// TIA Portal project "运动控制项目" (V20)

(* hardware
DEVICE "S7-1200 station_1"  S7-1200 Station
   slot 0: "Rack_0"  S7-1200 Rack  Rack  V1.0
   slot 1: "PLC_1"  CPU 1215C DC/DC/DC  6ES7 215-1AG40-0XB0  V4.6
   slot 3: "CB 1241 (RS485)"  CB 1241 (RS485)  6ES7 241-1CH30-1XB0  V1.0
*)

// ===== PLC "PLC_1"  CPU 1215C DC/DC/DC =====

VAR_GLOBAL   // PLC tag table "默认变量表"
   "System_Byte" AT %MB1 : Byte;
   "FirstScan" AT %M1.0 : Bool;
   "DiagStatusUpdate" AT %M1.1 : Bool;
   "AlwaysTRUE" AT %M1.2 : Bool;
   "AlwaysFALSE" AT %M1.3 : Bool;
   "Clock_Byte" AT %MB0 : Byte;
   "Clock_10Hz" AT %M0.0 : Bool;
   "Clock_5Hz" AT %M0.1 : Bool;
   "Clock_2.5Hz" AT %M0.2 : Bool;
   "Clock_2Hz" AT %M0.3 : Bool;
   "Clock_1.25Hz" AT %M0.4 : Bool;
   "Clock_1Hz" AT %M0.5 : Bool;
   "Clock_0.625Hz" AT %M0.6 : Bool;
   "Clock_0.5Hz" AT %M0.7 : Bool;
   "Tag_1" AT %Q0.6 : Bool;
   "Tag_2" AT %I0.3 : Bool;
   "Tag_3" AT %I0.4 : Bool;
   "Tag_4" AT %I0.5 : Bool;
   "Tag_5" AT %I0.6 : Bool;
   "Tag_6" AT %I0.7 : Bool;
   "Tag_7" AT %M2.4 : Bool;
   "Tag_8" AT %M2.5 : Bool;
END_VAR

VAR_GLOBAL   // PLC tag table "input"
   "limit_left" AT %I0.0 : Bool;
   "stop" AT %I0.1 : Bool;
   "limit_right" AT %I0.2 : Bool;
   "Tag_9" AT %I0.3 : Bool;
END_VAR

VAR_GLOBAL   // PLC tag table "output"
   "puls_plus" AT %Q0.0 : Bool;
   "red_w" AT %Q0.1 : Bool;
   "dir_plus" AT %Q0.2 : Bool;
   "green_s" AT %Q0.3 : Bool;
   "red_s" AT %Q0.4 : Bool;
   "yellow_s" AT %Q0.5 : Bool;
END_VAR

VAR_GLOBAL   // PLC tag table "intermedia"
   "cnt" AT %MB5 : Byte;
   "p1" AT %M2.0 : Bool;
   "p2" AT %M2.1 : Bool;
   "activate_x" AT %M2.2 : Bool;
   "ready_x" AT %M2.3 : Bool;
END_VAR

DATA_BLOCK "丝杠运动控制测试数据块_1"   // DB4
{ S7_Optimized_Access := 'TRUE' }
VERSION : 0.1
// stored: InstanceOfName 丝杠运动控制测试
"丝杠运动控制测试"
BEGIN
END_DATA_BLOCK

DATA_BLOCK "喷泉fc"   // DB5
{ S7_Optimized_Access := 'TRUE' }
VERSION : 0.1
BEGIN
END_DATA_BLOCK

// folder: 作业

DATA_BLOCK "交通红绿灯_流程SCL_DB"   // DB2
{ S7_Optimized_Access := 'TRUE' }
VERSION : 0.1
// stored: InstanceOfName 交通红绿灯_流程SCL
"交通红绿灯_流程SCL"
BEGIN
END_DATA_BLOCK

DATA_BLOCK "交通红绿灯_比较SCL_DB"   // DB3
{ S7_Optimized_Access := 'TRUE' }
VERSION : 0.1
// stored: InstanceOfName 交通红绿灯_比较SCL
"交通红绿灯_比较SCL"
BEGIN
END_DATA_BLOCK

// folder: (top level)

DATA_BLOCK "桌面丝杠"   // DB1, Motion_DB
{ S7_Optimized_Access := 'TRUE' }
AUTHOR : SIMATIC
FAMILY : BasicMC
NAME : TO_PosAx
VERSION : 8.0
// stored: InstanceOfName TO_PositioningAxis
"TO_PositioningAxis"
BEGIN
   // Axis.EnableOutput_AddressCU = %M2.2
   // Axis.PassiveHomingReferencePointSwitch_AddressCU = %I0.1
   // Axis.HomingReferencePointSwitch_AddressCU = %I0.1
   // Axis.PositionLimitsMin_AddressCU = %I0.0
   // Axis.PositionLimitsMax_AddressCU = %I0.2
   // Axis.OnlinePtoModeCU = 16#0000_0002
   // Axis.DirectionOutputEnabledCU = TRUE
   // Axis.SelectedChannel2EnumCU = %Q0.2
   // Axis.SelectedChannel1EnumCU = %Q0.0
   // Pulse.MinDeltaDeltaFrequencyCU = 0.004
   // Pulse.MaxDeltaDeltaFrequencyCU = 1.0E+10
   // Pulse.MinDeltaFrequencyCU = 0.005
   // Pulse.MaxDeltaFrequencyCU = 9.5E+9
   // Pulse.MinFrequencyCU = 1.0
   // Pulse.MaxFrequencyCU = 100000.0
   // Pulse.OutputSourceCU = 16#0000_0000
   // Axis.SelectPTO = 0
END_DATA_BLOCK

FUNCTION_BLOCK "丝杠运动控制测试"   // FB1, LAD
{ S7_Optimized_Access := 'TRUE' }
VERSION : 0.1
   VAR
      if_done : Bool;
      if_error : Bool;
      if_busy : Bool;
      error_id : Word;
      error_info : Word;
      ativate_x : Bool;
      ready_x : Bool;
      run_axis_x : Bool;
      position_x : DInt;
      MC_Power_Instance : MC_Power;
      MC_Home_Instance : MC_Home;
      MC_Power_Instance_1 : MC_Power;
      MC_ReadParam_Instance : MC_ReadParam;
      MC_WriteParam_Instance : MC_WriteParam;
      MC_MoveAbsolute_Instance : MC_MoveAbsolute;
      MC_MoveJog_Instance : MC_MoveJog;
      MC_Reset_Instance : MC_Reset;
   END_VAR
BEGIN

REGION Network 1
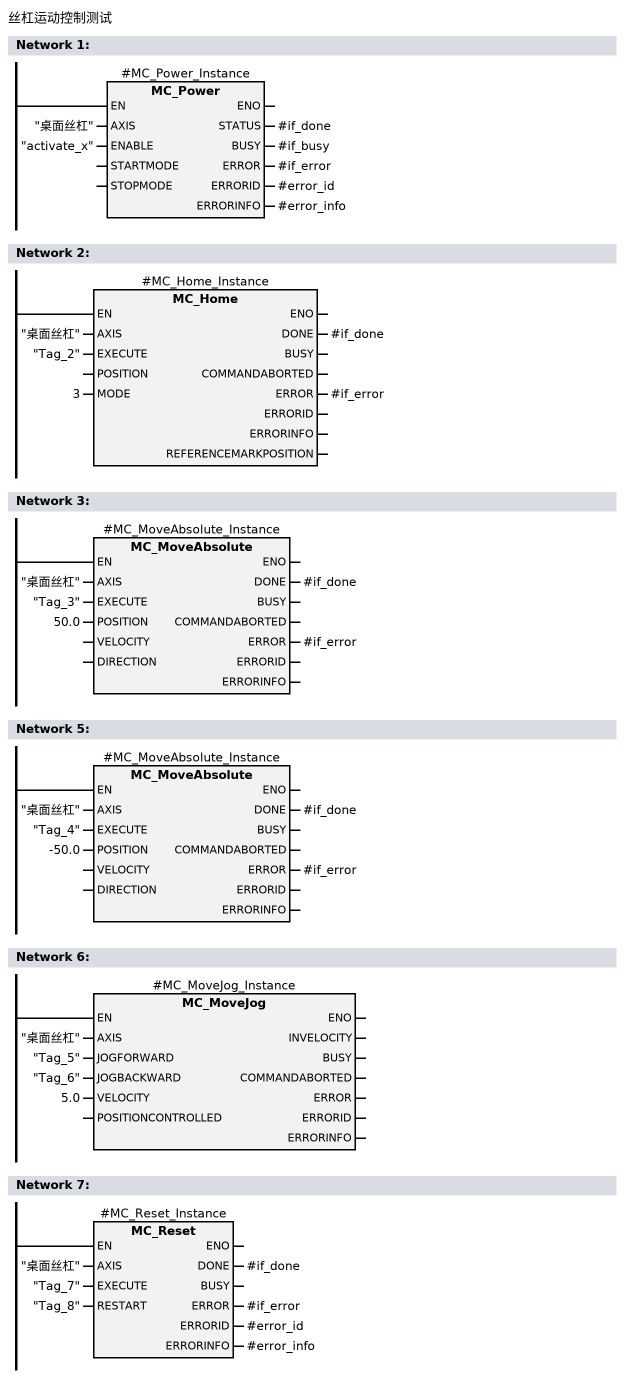
   #MC_Power_Instance(Axis := "桌面丝杠",   // MC_Power
                      Enable := "activate_x",
                      Status => #if_done,
                      Busy => #if_busy,
                      Error => #if_error,
                      ErrorID => #error_id,
                      ErrorInfo => #error_info);
END_REGION

REGION Network 2
   #MC_Home_Instance(Axis := "桌面丝杠", Execute := "Tag_2", Mode := 3, Done => #if_done, Error => #if_error);   // MC_Home
END_REGION

REGION Network 3
   #MC_MoveAbsolute_Instance(Axis := "桌面丝杠",   // MC_MoveAbsolute
                           Execute := "Tag_3",
                           Position := 50.0,
                           Done => #if_done,
                           Error => #if_error);
END_REGION

REGION Network 5
   #MC_MoveAbsolute_Instance(Axis := "桌面丝杠",   // MC_MoveAbsolute
                           Execute := "Tag_4",
                           Position := -50.0,
                           Done => #if_done,
                           Error => #if_error);
END_REGION

REGION Network 6
   #MC_MoveJog_Instance(Axis := "桌面丝杠", JogForward := "Tag_5", JogBackward := "Tag_6", Velocity := 5.0);   // MC_MoveJog
END_REGION

REGION Network 7
   #MC_Reset_Instance(Axis := "桌面丝杠",   // MC_Reset
                      Execute := "Tag_7",
                      Restart := "Tag_8",
                      Done => #if_done,
                      Error => #if_error,
                      ErrorID => #error_id,
                      ErrorInfo => #error_info);
END_REGION
END_FUNCTION_BLOCK

FUNCTION "喷泉项目" : Void   // FC2, LAD
{ S7_Optimized_Access := 'TRUE' }
VERSION : 0.1
BEGIN
END_FUNCTION

ORGANIZATION_BLOCK "Main"   // OB1, LAD, ProgramCycle
TITLE = "Main Program Sweep (Cycle)"
{ S7_Optimized_Access := 'TRUE' }
VERSION : 0.1
   VAR_INPUT
      Initial_Call : Bool;   // Initial call of this OB
      Remanence : Bool;   // =True, if remanent data are available
   END_VAR
BEGIN

REGION Network 1 (SCL)
   (*



   *)
END_REGION

REGION Network 2
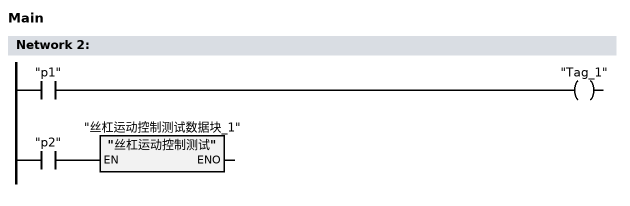
   RUNG wire#powerrail
      Contact( "p1" )
      Coil( "Tag_1" )
   END_RUNG
   RUNG wire#powerrail
      Contact( "p2" )
      "丝杠运动控制测试数据块_1"()
   END_RUNG
   // the same network as SCL:
   "Tag_1" := "p1";
   IF "p2" THEN
       "丝杠运动控制测试数据块_1"();   // "丝杠运动控制测试"
   END_IF;
END_REGION
END_ORGANIZATION_BLOCK

// folder: 作业

FUNCTION_BLOCK "交通红绿灯_流程SCL"   // FB2, LAD
{ S7_Optimized_Access := 'TRUE' }
VERSION : 0.1
   VAR
      start_pressed_trig : R_TRIG;
      stop_pressed_trig : R_TRIG;
      start_trig : R_TRIG;
      started : Bool;
      stoped : Bool;
      step_w : Byte;
      step_s : Byte;
      Timer_0 : TON_TIME;
      Timer_1 : TON_TIME;
      Timer_2 : TON_TIME;
      Timer_3 : TON_TIME;
      time_w : Time;
      time_s : Time;
   END_VAR
BEGIN

REGION Network 2 (SCL)
   IF "FirstScan" THEN
       #started := #stoped := 0;
       #step_w := #step_s := 0;
   END_IF;

   //initiate
   #start_pressed_trig(CLK := "limit_left");
   #stop_pressed_trig(CLK := "stop");
   #start_trig(CLK := #started);

   #Timer_0(IN := #started, PT := #time_w);
   #Timer_1(IN := #started, PT := #time_s);
   #Timer_2(IN := "AlwaysTRUE", PT := t#500ms);
   #Timer_3(IN := #Timer_2.Q,PT := t#500ms);
   IF #Timer_3.Q THEN
       RESET_TIMER(#Timer_2);
   END_IF;

   IF #start_pressed_trig.Q THEN
       #started := 1;
       #stoped := 0;
   END_IF;

   IF #start_trig.Q THEN
       #stoped := 0;
       #step_s := #step_w := 0;
       "green_s" := "puls_plus" := "dir_plus" := "yellow_s" := "red_w" := "red_s" := 0;
       #time_w := t#5s;
       #time_s := t#10s;
       RESET_TIMER(#Timer_0);
       RESET_TIMER(#Timer_1);
   END_IF;

   IF #stop_pressed_trig.Q THEN
       #stoped := 1;
   END_IF;

   IF #started THEN
       //东西向
       IF #step_w = 0 THEN
           "puls_plus" := 1;
           IF #Timer_0.Q THEN
               "puls_plus" := 0;
               RESET_TIMER(#Timer_0);
               #time_w := T#3s;
               #step_w += 1;
           END_IF;
       END_IF;

       IF #step_w = 1 THEN
           "puls_plus" := #Timer_2.Q;
           IF #Timer_0.Q THEN
               "puls_plus" := 0;
               RESET_TIMER(#Timer_0);
               #time_w := T#2s;
               #step_w += 1;
           END_IF;
       END_IF;

       IF #step_w = 2 THEN
           "dir_plus" := 1;
           IF #Timer_0.Q THEN
               "dir_plus" := 0;
               RESET_TIMER(#Timer_0);
               #time_w := T#10s;
               #step_w += 1;
           END_IF;
       END_IF;

       IF #step_w = 3 THEN
           "red_w":= 1;
           IF #Timer_0.Q THEN
               "red_w" := 0;
               RESET_TIMER(#Timer_0);
               #time_w := T#5s;
               #step_w := 0;
           END_IF;
       END_IF;

       //南北向
       IF #step_s = 0 THEN
           "red_s" := 1;
           IF #Timer_1.Q THEN
               "red_s" := 0;
               RESET_TIMER(#Timer_1);
               #time_s := T#5s;
               #step_s += 1;
           END_IF;
       END_IF;

       IF #step_s = 1 THEN
           "green_s" := 1;
           IF #Timer_1.Q THEN
               "green_s" := 0;
               RESET_TIMER(#Timer_1);
               #time_s := T#3s;
               #step_s += 1;
           END_IF;
       END_IF;

       IF #step_s = 2 THEN
          "green_s" := #Timer_2.Q;
          IF #Timer_1.Q THEN
              "green_s" := 0;
               RESET_TIMER(#Timer_1);
               #time_s := T#2s;
               #step_s += 1;
           END_IF;
       END_IF;

       IF #step_s = 3 THEN
           "yellow_s" := 1;
           IF #Timer_1.Q THEN
               "yellow_s" := 0;
               RESET_TIMER(#Timer_1);
               #time_s := T#10s;
               #step_s := 0;
               #step_w := 0;
               "red_w" := 0;
               RESET_TIMER(#Timer_0);
               #time_w := T#5s;
               #step_w := 0;

               IF #stoped THEN
                   #started := 0;
                   #stoped := 0;
               END_IF;
           END_IF;
       END_IF;
   END_IF;

   IF NOT #stoped AND NOT #started THEN
       "yellow_s" := #Timer_2.Q;
       "dir_plus" := #Timer_2.Q;
   END_IF;
END_REGION
END_FUNCTION_BLOCK

FUNCTION_BLOCK "交通红绿灯_比较SCL"   // FB3, LAD
{ S7_Optimized_Access := 'TRUE' }
VERSION : 0.1
   VAR
      start_pressed_trig : R_TRIG;
      stop_pressed_trig : R_TRIG;
      start_trig : R_TRIG;
      started : Bool;
      stoped : Bool;
      step_w : Byte;
      step_s : Byte;
      Timer_0 : TON_TIME;
      Timer_1 : TON_TIME;
      Timer_2 : TON_TIME;
      Timer_3 : TON_TIME;
      time_w : Time;
      time_s : Time;
      button : Array[0..10] of Bool;
      b1 : Bool;
      b2 : Bool;
      b4 : Bool;
      b3 : Bool;
      b5 : Bool;
   END_VAR
BEGIN

REGION Network 2 (SCL)
   IF "FirstScan" THEN
       #started := #stoped := 0;
       #step_w := #step_s := 0;
   END_IF;

   //initiate
   #start_pressed_trig(CLK := "limit_left");
   #stop_pressed_trig(CLK := "stop");
   #start_trig(CLK := #started);

   #Timer_0(IN := #started, PT := t#20S);
   #Timer_2(IN := "AlwaysTRUE", PT := t#500ms);
   #Timer_3(IN := #Timer_2.Q,PT := t#500ms);
   IF #Timer_3.Q THEN
       RESET_TIMER(#Timer_2);
   END_IF;

   IF #start_pressed_trig.Q THEN
       #started := 1;
       #stoped := 0;
   END_IF;

   IF #start_trig.Q THEN
       #stoped := 0;
       RESET_TIMER(#Timer_0);
       RESET_TIMER(#Timer_2);
   END_IF;

   IF #stop_pressed_trig.Q THEN
       #stoped := 1;
   END_IF;

   IF #started THEN
       //东西向
       "puls_plus" := #Timer_0.ET > t#0s AND #Timer_0.ET <= t#5s OR (#Timer_0.ET > t#5s AND #Timer_0.ET <= t#8s AND #Timer_2.Q);
       "dir_plus" := #Timer_0.ET > t#8s AND #Timer_0.ET <= t#10s;
       "red_w" := #Timer_0.ET > t#10s AND #Timer_0.ET <= t#20s;

       //南北向
       "red_s" := #Timer_0.ET > t#0s AND #Timer_0.ET <= t#10s;
       "green_s" := #Timer_0.ET > t#10s AND #Timer_0.ET <= t#13s OR (#Timer_0.ET > t#13s AND #Timer_0.ET <= t#15s AND #Timer_2.Q);
       "yellow_s" := #Timer_0.ET > t#15s AND #Timer_0.ET < t#20s;

       IF #Timer_0.ET >= t#20S THEN
           RESET_TIMER(#Timer_0);
           RESET_TIMER(#Timer_1);

           #started := NOT #stoped;
           #stoped := 0;
       END_IF;
   END_IF;

   IF NOT #stoped AND NOT #started THEN
       "green_s" := "puls_plus" := "red_s" := "red_w" := 0;
       "yellow_s" := #Timer_2.Q;
       "dir_plus" := #Timer_2.Q;
   END_IF;
END_REGION
END_FUNCTION_BLOCK

FUNCTION "红绿灯_FC" : Void   // FC1, LAD
{ S7_Optimized_Access := 'TRUE' }
VERSION : 0.1
   VAR_TEMP   // added for the SCL form of the ladder/FBD networks
      _w1 : Bool;
      _w2 : Bool;
      _w3 : Bool;
   END_VAR
BEGIN

REGION Network 1
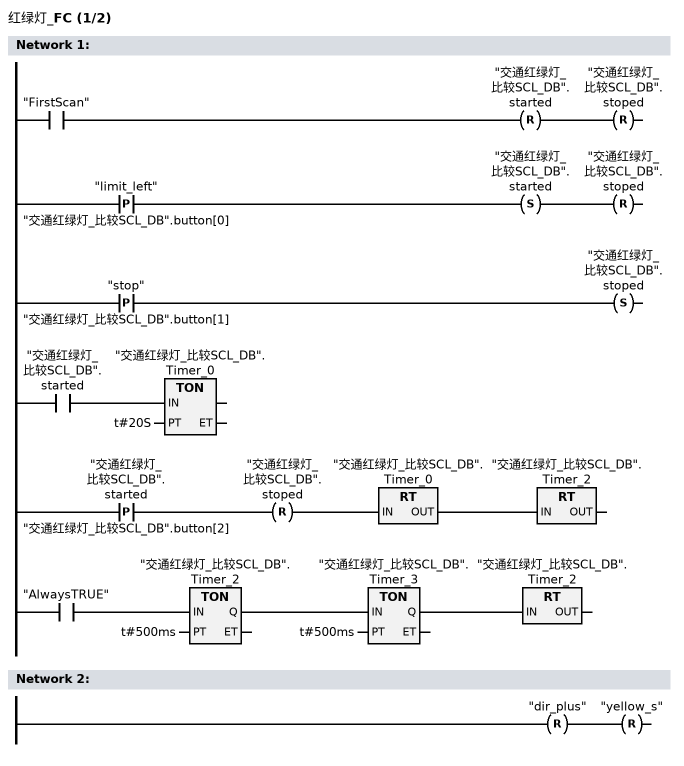
   IF "FirstScan" THEN
       "交通红绿灯_比较SCL_DB".started := FALSE;
       "交通红绿灯_比较SCL_DB".stoped := FALSE;
   END_IF;
   #_w1 := "limit_left" AND NOT "交通红绿灯_比较SCL_DB".button[0];   // rising edge of "limit_left"
   "交通红绿灯_比较SCL_DB".button[0] := "limit_left";
   IF #_w1 THEN
       "交通红绿灯_比较SCL_DB".started := TRUE;
       "交通红绿灯_比较SCL_DB".stoped := FALSE;
   END_IF;
   #_w2 := "stop" AND NOT "交通红绿灯_比较SCL_DB".button[1];   // rising edge of "stop"
   "交通红绿灯_比较SCL_DB".button[1] := "stop";
   IF #_w2 THEN "交通红绿灯_比较SCL_DB".stoped := TRUE; END_IF;
   "交通红绿灯_比较SCL_DB".Timer_0.TON(IN := "交通红绿灯_比较SCL_DB".started, PT := t#20S);
   #_w3 := "交通红绿灯_比较SCL_DB".started AND NOT "交通红绿灯_比较SCL_DB".button[2];   // rising edge of "交通红绿灯_比较SCL_DB".started
   "交通红绿灯_比较SCL_DB".button[2] := "交通红绿灯_比较SCL_DB".started;
   IF #_w3 THEN
       "交通红绿灯_比较SCL_DB".stoped := FALSE;
       RESET_TIMER("交通红绿灯_比较SCL_DB".Timer_0);
       RESET_TIMER("交通红绿灯_比较SCL_DB".Timer_2);
   END_IF;
   "交通红绿灯_比较SCL_DB".Timer_2.TON(IN := "AlwaysTRUE", PT := t#500ms);
   "交通红绿灯_比较SCL_DB".Timer_3.TON(IN := "交通红绿灯_比较SCL_DB".Timer_2.Q, PT := t#500ms);
   IF "交通红绿灯_比较SCL_DB".Timer_3.Q THEN RESET_TIMER("交通红绿灯_比较SCL_DB".Timer_2); END_IF;
END_REGION

REGION Network 2
   RUNG wire#powerrail
      R_Coil( "dir_plus" )
      R_Coil( "yellow_s" )
   END_RUNG
   // the same network as SCL:
   "dir_plus" := FALSE;
   "yellow_s" := FALSE;
END_REGION

REGION Network 3
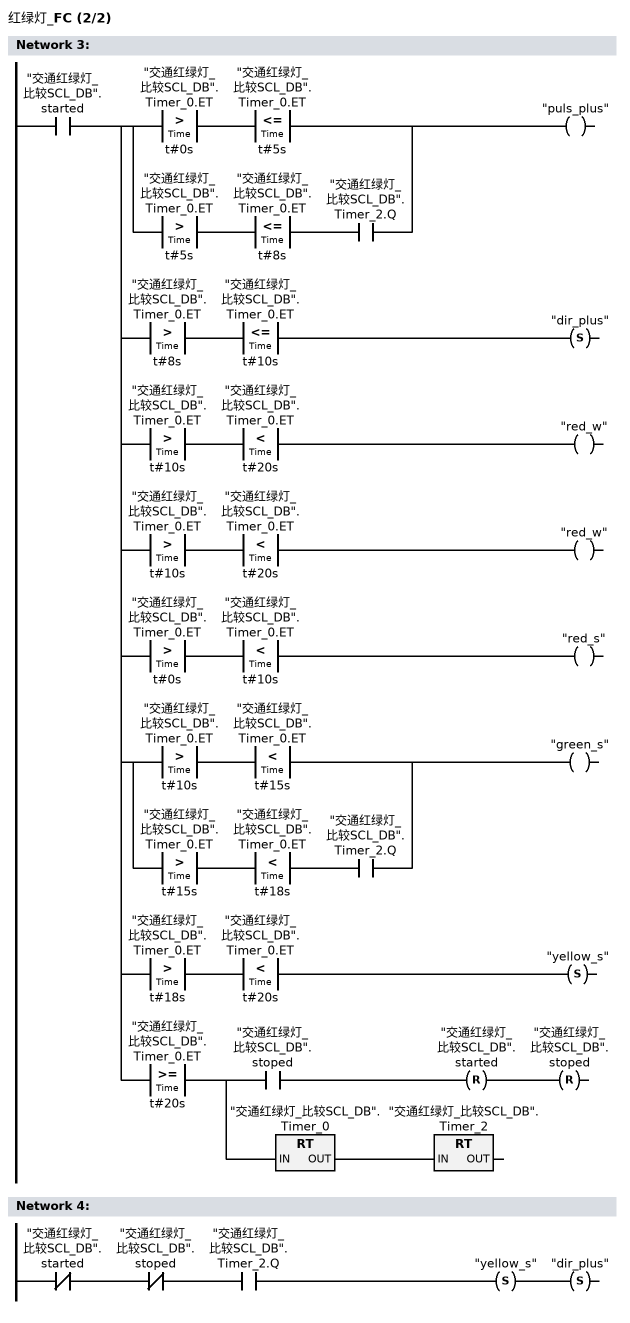
   RUNG wire#powerrail
      Contact( "交通红绿灯_比较SCL_DB".started )
      wire#w1
      { S7_Templates := "SrcType := Time" } GT_Contact(in1 := "交通红绿灯_比较SCL_DB".Timer_0.ET, in2 := t#0s)
      { S7_Templates := "SrcType := Time" } LE_Contact(in1 := "交通红绿灯_比较SCL_DB".Timer_0.ET, in2 := t#5s)
      wire#w2
      Coil( "puls_plus" )
   END_RUNG
   RUNG wire#w1
      { S7_Templates := "SrcType := Time" } GT_Contact(in1 := "交通红绿灯_比较SCL_DB".Timer_0.ET, in2 := t#5s)
      { S7_Templates := "SrcType := Time" } LE_Contact(in1 := "交通红绿灯_比较SCL_DB".Timer_0.ET, in2 := t#8s)
      Contact( "交通红绿灯_比较SCL_DB".Timer_2.Q )
   END_RUNG wire#w2
   RUNG wire#w1
      { S7_Templates := "SrcType := Time" } GT_Contact(in1 := "交通红绿灯_比较SCL_DB".Timer_0.ET, in2 := t#8s)
      { S7_Templates := "SrcType := Time" } LE_Contact(in1 := "交通红绿灯_比较SCL_DB".Timer_0.ET, in2 := t#10s)
      S_Coil( "dir_plus" )
   END_RUNG
   RUNG wire#w1
      { S7_Templates := "SrcType := Time" } GT_Contact(in1 := "交通红绿灯_比较SCL_DB".Timer_0.ET, in2 := t#10s)
      { S7_Templates := "SrcType := Time" } LT_Contact(in1 := "交通红绿灯_比较SCL_DB".Timer_0.ET, in2 := t#20s)
      Coil( "red_w" )
   END_RUNG
   RUNG wire#w1
      { S7_Templates := "SrcType := Time" } GT_Contact(in1 := "交通红绿灯_比较SCL_DB".Timer_0.ET, in2 := t#10s)
      { S7_Templates := "SrcType := Time" } LT_Contact(in1 := "交通红绿灯_比较SCL_DB".Timer_0.ET, in2 := t#20s)
      Coil( "red_w" )
   END_RUNG
   RUNG wire#w1
      { S7_Templates := "SrcType := Time" } GT_Contact(in1 := "交通红绿灯_比较SCL_DB".Timer_0.ET, in2 := t#0s)
      { S7_Templates := "SrcType := Time" } LT_Contact(in1 := "交通红绿灯_比较SCL_DB".Timer_0.ET, in2 := t#10s)
      Coil( "red_s" )
   END_RUNG
   RUNG wire#w1
      { S7_Templates := "SrcType := Time" } GT_Contact(in1 := "交通红绿灯_比较SCL_DB".Timer_0.ET, in2 := t#10s)
      { S7_Templates := "SrcType := Time" } LT_Contact(in1 := "交通红绿灯_比较SCL_DB".Timer_0.ET, in2 := t#15s)
      wire#w3
      Coil( "green_s" )
   END_RUNG
   RUNG wire#w1
      { S7_Templates := "SrcType := Time" } GT_Contact(in1 := "交通红绿灯_比较SCL_DB".Timer_0.ET, in2 := t#15s)
      { S7_Templates := "SrcType := Time" } LT_Contact(in1 := "交通红绿灯_比较SCL_DB".Timer_0.ET, in2 := t#18s)
      Contact( "交通红绿灯_比较SCL_DB".Timer_2.Q )
   END_RUNG wire#w3
   RUNG wire#w1
      { S7_Templates := "SrcType := Time" } GT_Contact(in1 := "交通红绿灯_比较SCL_DB".Timer_0.ET, in2 := t#18s)
      { S7_Templates := "SrcType := Time" } LT_Contact(in1 := "交通红绿灯_比较SCL_DB".Timer_0.ET, in2 := t#20s)
      S_Coil( "yellow_s" )
   END_RUNG
   RUNG wire#w1
      { S7_Templates := "SrcType := Time" } GE_Contact(in1 := "交通红绿灯_比较SCL_DB".Timer_0.ET, in2 := t#20s)
      wire#w4
      Contact( "交通红绿灯_比较SCL_DB".stoped )
      R_Coil( "交通红绿灯_比较SCL_DB".started )
      R_Coil( "交通红绿灯_比较SCL_DB".stoped )
   END_RUNG
   RUNG wire#w4
      RT_Coil( "交通红绿灯_比较SCL_DB".Timer_0 )
      RT_Coil( "交通红绿灯_比较SCL_DB".Timer_2 )
   END_RUNG
   // the same network as SCL:
   "puls_plus" := "交通红绿灯_比较SCL_DB".started AND ((("交通红绿灯_比较SCL_DB".Timer_0.ET > t#0s) AND ("交通红绿灯_比较SCL_DB".Timer_0.ET <= t#5s)) OR (("交通红绿灯_比较SCL_DB".Timer_0.ET > t#5s) AND ("交通红绿灯_比较SCL_DB".Timer_0.ET <= t#8s) AND "交通红绿灯_比较SCL_DB".Timer_2.Q));
   IF "交通红绿灯_比较SCL_DB".started AND ("交通红绿灯_比较SCL_DB".Timer_0.ET > t#8s) AND ("交通红绿灯_比较SCL_DB".Timer_0.ET <= t#10s) THEN
       "dir_plus" := TRUE;
   END_IF;
   "red_w" := "交通红绿灯_比较SCL_DB".started AND ("交通红绿灯_比较SCL_DB".Timer_0.ET > t#10s) AND ("交通红绿灯_比较SCL_DB".Timer_0.ET < t#20s);
   "red_w" := "交通红绿灯_比较SCL_DB".started AND ("交通红绿灯_比较SCL_DB".Timer_0.ET > t#10s) AND ("交通红绿灯_比较SCL_DB".Timer_0.ET < t#20s);
   "red_s" := "交通红绿灯_比较SCL_DB".started AND ("交通红绿灯_比较SCL_DB".Timer_0.ET > t#0s) AND ("交通红绿灯_比较SCL_DB".Timer_0.ET < t#10s);
   "green_s" := "交通红绿灯_比较SCL_DB".started AND ((("交通红绿灯_比较SCL_DB".Timer_0.ET > t#10s) AND ("交通红绿灯_比较SCL_DB".Timer_0.ET < t#15s)) OR (("交通红绿灯_比较SCL_DB".Timer_0.ET > t#15s) AND ("交通红绿灯_比较SCL_DB".Timer_0.ET < t#18s) AND "交通红绿灯_比较SCL_DB".Timer_2.Q));
   IF "交通红绿灯_比较SCL_DB".started AND ("交通红绿灯_比较SCL_DB".Timer_0.ET > t#18s) AND ("交通红绿灯_比较SCL_DB".Timer_0.ET < t#20s) THEN
       "yellow_s" := TRUE;
   END_IF;
   #_w1 := "交通红绿灯_比较SCL_DB".started AND ("交通红绿灯_比较SCL_DB".Timer_0.ET >= t#20s);
   IF #_w1 AND "交通红绿灯_比较SCL_DB".stoped THEN
       "交通红绿灯_比较SCL_DB".started := FALSE;
       "交通红绿灯_比较SCL_DB".stoped := FALSE;
   END_IF;
   IF #_w1 THEN
       RESET_TIMER("交通红绿灯_比较SCL_DB".Timer_0);
       RESET_TIMER("交通红绿灯_比较SCL_DB".Timer_2);
   END_IF;
END_REGION

REGION Network 4
   RUNG wire#powerrail
      I_Contact( "交通红绿灯_比较SCL_DB".started )
      I_Contact( "交通红绿灯_比较SCL_DB".stoped )
      Contact( "交通红绿灯_比较SCL_DB".Timer_2.Q )
      S_Coil( "yellow_s" )
      S_Coil( "dir_plus" )
   END_RUNG
   // the same network as SCL:
   IF NOT "交通红绿灯_比较SCL_DB".started AND NOT "交通红绿灯_比较SCL_DB".stoped AND "交通红绿灯_比较SCL_DB".Timer_2.Q THEN
       "yellow_s" := TRUE;
       "dir_plus" := TRUE;
   END_IF;
END_REGION
END_FUNCTION